FUNCTION_BLOCK BYPASS (* Bypass FB *)
  (* Standard: 61499-2 *)
  (* Version 1.0, 2026-05-07, franz *)
  PACKAGE logiBUS::signalprocessing::bypass;
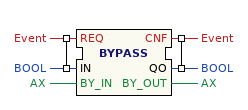
  EVENT_INPUT
    REQ WITH IN; (* Normal Execution Request *)
  END_EVENT
  EVENT_OUTPUT
    CNF WITH QO; (* Execution Confirmation *)
  END_EVENT
  VAR_INPUT
    IN : BOOL; (* Input *)
  END_VAR
  VAR_OUTPUT
    QO : BOOL; (* Output *)
  END_VAR
  SOCKETS
    BY_IN : adapter::types::unidirectional::AX; (* Bypass in *)
  END_SOCKETS
  PLUGS
    BY_OUT : adapter::types::unidirectional::AX; (* Bypass out *)
  END_PLUGS
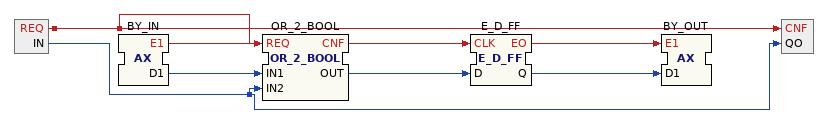
  FBS
    OR_2_BOOL : iec61131::bitwiseOperators::OR_2_BOOL;
    E_D_FF : iec61499::events::E_D_FF;
  END_FBS
  EVENT_CONNECTIONS
    OR_2_BOOL.CNF TO E_D_FF.CLK;
    BY_IN.E1 TO OR_2_BOOL.REQ;
    E_D_FF.EO TO BY_OUT.E1;
    REQ TO CNF;
    REQ TO OR_2_BOOL.REQ;
  END_CONNECTIONS
  DATA_CONNECTIONS
    OR_2_BOOL.OUT TO E_D_FF.D;
    BY_IN.D1 TO OR_2_BOOL.IN1;
    E_D_FF.Q TO BY_OUT.D1;
    IN TO OR_2_BOOL.IN2;
    IN TO QO;
  END_CONNECTIONS
END_FUNCTION_BLOCK
